// TwinCAT 3 PLC project Sample01
// ProgramVersion: 3.1.4022.1
// libraries:
//   Tc2_Standard, * (Beckhoff Automation GmbH)
//   Tc2_System, * (Beckhoff Automation GmbH)
//   Tc3_Module, * (Beckhoff Automation GmbH)
// project tree:
//   GVLs/ Param.TcGVL
//   / PlcTask.TcTTO
//   POUs/ FB_Observer.TcPOU, FB_Subject.TcPOU, MAIN.TcPOU, I_Observer.TcIO, I_Subject.TcIO
// real-time tasks:
//   TASK PlcTask: cycle T#10ms, priority 20, ADS port 350

CONFIGURATION Sample01
    RESOURCE PLC ON TwinCAT3
        TASK PlcTask(INTERVAL := T#10ms, PRIORITY := 20);
        PROGRAM MAIN WITH PlcTask : MAIN;
    END_RESOURCE
END_CONFIGURATION

// ---- GVLs/Param.TcGVL
{attribute 'qualified_only'}
VAR_GLOBAL CONSTANT
	// size of the observer array
	cMaxObservers		: INT := 10;	
END_VAR

// ---- POUs/I_Observer.TcIO
INTERFACE I_Observer

METHOD Update
VAR_INPUT	
	fValue			: LREAL;
END_VAR
END_METHOD

END_INTERFACE

// ---- POUs/I_Subject.TcIO
INTERFACE I_Subject

METHOD Attach : BOOL
VAR_INPUT
	ipObserver		: I_Observer;
END_VAR
END_METHOD

METHOD Detach : BOOL
VAR_INPUT	
	ipObserver		: I_Observer;
END_VAR
END_METHOD

END_INTERFACE

// ---- POUs/MAIN.TcPOU
PROGRAM MAIN
VAR
	fbSubject 			: FB_Subject;
	fbObserver1 		: FB_Observer;
	fbObserver2 		: FB_Observer;
	
	bAttachObserver1	: BOOL;
	bAttachObserver2	: BOOL;

	bDetachObserver1	: BOOL;
	bDetachObserver2	: BOOL;
END_VAR

fbSubject();

IF (bAttachObserver1) THEN
	fbSubject.Attach(fbObserver1);
	bAttachObserver1 := FALSE;
END_IF

IF (bAttachObserver2) THEN
	fbSubject.Attach(fbObserver2);
	bAttachObserver2 := FALSE;
END_IF

IF (bDetachObserver1) THEN
	fbSubject.Detach(fbObserver1);
	bDetachObserver1 := FALSE;
END_IF

IF (bDetachObserver2) THEN
	fbSubject.Detach(fbObserver2);
	bDetachObserver2 := FALSE;
END_IF

END_PROGRAM

// ---- POUs/FB_Subject.TcPOU
FUNCTION_BLOCK PUBLIC FB_Subject IMPLEMENTS I_Subject
VAR	
	fbDelay				: TON;
	fbDrand				: DRAND;
	fValue				: LREAL;
	aObservers			: ARRAY [1..Param.cMaxObservers] OF I_Observer;
END_VAR

// creates every sec a random value and invoke the update method
fbDelay(IN := TRUE, PT := T#1S);
IF (fbDelay.Q) THEN	
	fbDelay(IN := FALSE);	
	fbDrand(SEED := 0);
	fValue := fbDrand.Num * 1234.5;
	Notify();
END_IF

METHOD PUBLIC Attach : BOOL
VAR_INPUT
	ipObserver				: I_Observer;
END_VAR
VAR
	nIndex					: INT := 0;
END_VAR
Attach := FALSE;
IF (ipObserver = 0) THEN
	RETURN;
END_IF

// is the observer already registered?
FOR nIndex := 1 TO Param.cMaxObservers DO	
	IF (THIS^.aObservers[nIndex] = ipObserver) THEN
		RETURN;
	END_IF
END_FOR

// save the observer object into the array of observers and send the actual value
FOR nIndex := 1 TO Param.cMaxObservers DO
	IF (THIS^.aObservers[nIndex] = 0) THEN
		THIS^.aObservers[nIndex] := ipObserver;
		THIS^.aObservers[nIndex].Update(THIS^.fValue);
		Attach := TRUE;
		EXIT;					
	END_IF
END_FOR
END_METHOD

METHOD PUBLIC Detach : BOOL
VAR_INPUT
	ipObserver		: I_Observer;
END_VAR
VAR
	nIndex			: INT := 0;
END_VAR
Detach := FALSE;
IF (ipObserver = 0) THEN
	RETURN;
END_IF

FOR nIndex := 1 TO Param.cMaxObservers DO
	IF (THIS^.aObservers[nIndex] = ipObserver) THEN
		THIS^.aObservers[nIndex] := 0;
		Detach := TRUE;	
	END_IF
END_FOR
END_METHOD

{attribute 'monitoring':='call'}
PROPERTY PUBLIC fActualValue : LREAL
GET
fActualValue := THIS^.fValue;
END_GET
END_PROPERTY

METHOD PRIVATE Notify
VAR	
	nIndex		: INT := 0;
END_VAR
FOR nIndex := 1 TO Param.cMaxObservers DO
	IF (THIS^.aObservers[nIndex] <> 0) THEN
		THIS^.aObservers[nIndex].Update(THIS^.fActualValue);
	END_IF
END_FOR
END_METHOD

END_FUNCTION_BLOCK

// ---- POUs/FB_Observer.TcPOU
FUNCTION_BLOCK PUBLIC FB_Observer IMPLEMENTS I_Observer
VAR
	fValue				: LREAL;
END_VAR

{attribute 'monitoring':='call'}
PROPERTY PUBLIC fActualValue : LREAL
GET
fActualValue := THIS^.fValue;
END_GET
END_PROPERTY

METHOD PUBLIC Update
VAR_INPUT
	fValue			: LREAL;
END_VAR
THIS^.fValue := fValue;
END_METHOD

END_FUNCTION_BLOCK
